Staubli VAL3: HIT_YD.pjx

--- HIT_YD.pjx ---
Parameters version=s7.6.4 stackSize=5000 millimeterUnit=true
Program file=blow.pgx
Program file=bypassPick.pgx
Program file=cellManager.pgx
Program file=getToolStatus.pgx
Program file=goHome.pgx
Program file=init.pgx
Program file=initTracking.pgx
Program file=isInSafetyArea.pgx
Program file=modbusGet.pgx
Program file=modbusSet.pgx
Program file=OMAC_Abort.pgx
Program file=OMAC_Hold.pgx
Program file=OMAC_Main.pgx
Program file=OMAC_Reset.pgx
Program file=OMAC_Start.pgx
Program file=OMAC_Stop.pgx
Program file=OMAC_Unhold.pgx
Program file=overflowPick.pgx
Program file=Place.pgx
Program file=productionCycle.pgx
Program file=robot2PLC.pgx
Program file=send2NextRob.pgx
Program file=setAlarm.pgx
Program file=setConvSpeed.pgx
Program file=start.pgx
Program file=stop.pgx
Program file=trackErr_init.pgx
Program file=trackingPick.pgx
Program file=transferQueue.pgx
Data file=HIT_YD.dtx
Library alias=mot path=Disk://Tracking/Motion/Motion.pjx
Type name=object path=Disk://Tracking/Templates/object/object.pjx

--- init.pgx ---
program init()
  local num l_nI
  local num l_nJ
begin
  // This program initialize all variables
  //
  // Input parameters
  //  None            :
  //
  // Output parameters
  //  None            :
  //
  //----------------------------------------------------------------
  //
  //che add
  nPlaceNum=0
  // Booleans
  _bSentToHome=false
  _bMutexCnvQueue[0]=false
  _bIsPicking=false
  _bIsPlacing=false
  _bConvExist=false
  _bEndCycle=false
  //

  //
  // Numerical
  _nBlowDelay=0
  _nID[0]=-1
  _nCntBypassed[0]=nBypass[0]
  _nCntTransfered[0]=0

  _nPushIndexTQ[0]=0
  _nPullIndexTQ[0]=0
  _nTimer=0

  resize(_nCycleTime,1,4)
  for _nCycleTimeIndx=0 to size(_nCycleTime)-1
    _nCycleTime[_nCycleTimeIndx]=0
  endFor
  _nCycleTimeIndx=0

  //dio
  dPlaceDone[0]=false
  dPlaceDone[1]=false
  dPlaceDone[2]=false
  dPlaceDone[3]=false

  // aio
  aioSet(aRbAlarm,0)
  //call setAlarm(0)

  clearBuffer(toRobot1)
  // Points
  pPick.trsf={0,0,0,0,0,0}

  //

  //
  // Transfer Queues
  for l_nI=0 to size(_oTransferQueue,2)-1
    _oTransferQueue[0,l_nI].nID=-1
    _oTransferQueue[0,l_nI].trTrsf={0,0,0,0,0,0}
    _oTransferQueue[0,l_nI].nLatchedValue=0
  endFor
  //
  // Strings
  _sCycleStatus=""
  autoConnectMove(true)
end

--- setAlarm.pgx ---
program setAlarm(num x_nNum)
begin
  switch x_nNum
    case 0
      dAlarm[0]=true
      dAlarm[1]=false
      dAlarm[2]=false
      dAlarm[3]=false
      dAlarm[4]=false
      dAlarm[5]=false
      dAlarm[6]=false
      dAlarm[7]=false
      delay(0.35)
      dAlarm[0]=false
      dAlarm[1]=false
      dAlarm[2]=false
      dAlarm[3]=false
      dAlarm[4]=false
      dAlarm[5]=false
      dAlarm[6]=false
      dAlarm[7]=false
    break
    case 1
      dAlarm[0]=false
      dAlarm[1]=true
      dAlarm[2]=false
      dAlarm[3]=false
      dAlarm[4]=false
      dAlarm[5]=false
      dAlarm[6]=false
      dAlarm[7]=false
      delay(0.35)
      dAlarm[0]=false
      dAlarm[1]=false
      dAlarm[2]=false
      dAlarm[3]=false
      dAlarm[4]=false
      dAlarm[5]=false
      dAlarm[6]=false
      dAlarm[7]=false
    break
    case 2
      dAlarm[0]=false
      dAlarm[1]=false
      dAlarm[2]=true
      dAlarm[3]=false
      dAlarm[4]=false
      dAlarm[5]=false
      dAlarm[6]=false
      dAlarm[7]=false
      delay(0.35)
      dAlarm[0]=false
      dAlarm[1]=false
      dAlarm[2]=false
      dAlarm[3]=false
      dAlarm[4]=false
      dAlarm[5]=false
      dAlarm[6]=false
      dAlarm[7]=false
    break
    case 3
      dAlarm[0]=false
      dAlarm[1]=false
      dAlarm[2]=true
      dAlarm[3]=false
      dAlarm[4]=false
      dAlarm[5]=false
      dAlarm[6]=false
      dAlarm[7]=false
      delay(0.35)
      dAlarm[0]=false
      dAlarm[1]=false
      dAlarm[2]=false
      dAlarm[3]=false
      dAlarm[4]=false
      dAlarm[5]=false
      dAlarm[6]=false
      dAlarm[7]=false
    break
    case 4
      dAlarm[0]=false
      dAlarm[1]=false
      dAlarm[2]=false
      dAlarm[3]=false
      dAlarm[4]=true
      dAlarm[5]=false
      dAlarm[6]=false
      dAlarm[7]=false
      delay(0.35)
      dAlarm[0]=false
      dAlarm[1]=false
      dAlarm[2]=false
      dAlarm[3]=false
      dAlarm[4]=false
      dAlarm[5]=false
      dAlarm[6]=false
      dAlarm[7]=false
    break
    case 5
      dAlarm[0]=false
      dAlarm[1]=false
      dAlarm[2]=false
      dAlarm[3]=false
      dAlarm[4]=false
      dAlarm[5]=true
      dAlarm[6]=false
      dAlarm[7]=false
      delay(0.35)
      dAlarm[0]=false
      dAlarm[1]=false
      dAlarm[2]=false
      dAlarm[3]=false
      dAlarm[4]=false
      dAlarm[5]=false
      dAlarm[6]=false
      dAlarm[7]=false
    break
    case 6
      dAlarm[0]=false
      dAlarm[1]=false
      dAlarm[2]=false
      dAlarm[3]=false
      dAlarm[4]=false
      dAlarm[5]=false
      dAlarm[6]=true
      dAlarm[7]=false
      delay(0.35)
      dAlarm[0]=false
      dAlarm[1]=false
      dAlarm[2]=false
      dAlarm[3]=false
      dAlarm[4]=false
      dAlarm[5]=false
      dAlarm[6]=false
      dAlarm[7]=false
    break
    case 7
      dAlarm[0]=false
      dAlarm[1]=false
      dAlarm[2]=false
      dAlarm[3]=false
      dAlarm[4]=false
      dAlarm[5]=false
      dAlarm[6]=false
      dAlarm[7]=true
      delay(0.35)
      dAlarm[0]=false
      dAlarm[1]=false
      dAlarm[2]=false
      dAlarm[3]=false
      dAlarm[4]=false
      dAlarm[5]=false
      dAlarm[6]=false
      dAlarm[7]=false
    break
    default
      dAlarm[0]=false
      dAlarm[1]=false
      dAlarm[2]=false
      dAlarm[3]=false
      dAlarm[4]=false
      dAlarm[5]=false
      dAlarm[6]=false
      dAlarm[7]=false
    break
  endSwitch
end

--- setConvSpeed.pgx ---
program setConvSpeed(num x_nConvNum (dimensions=1), num x_nConvSpeed (dimensions=1))
  local num l_nRatio[2]
begin
  // This programs sets, by an analog output, the speed of the
  //  conveyor. The program takes as an input parameter the speed in
  //  mm/s, then it will convert it to the corresponding value that
  //  has to be actually written into the analog output. The local
  //  variable l_nRatio has to be adapted to match the hardware.
  //
  // Input parameters
  //  x_nConvNum      : Conveyor number
  //  x_nConvSpeed    : Conveyor speed in mm/s
  //
  // Output parameters
  //  None            :
  //
  //----------------------------------------------------------------
  //
  l_nRatio[0]=35
  //
  if ioStatus(aConvSpeed[x_nConvNum])>=0
    aioSet(aConvSpeed[x_nConvNum],x_nConvSpeed*l_nRatio[x_nConvNum])
  endIf
  //
end
